fb_derevo_vidpochynok1_send(str_Rec:=fb_KL6301_0.str_Data_Rec, bData:=derevo_vidpochynok1,  Group_Address:=derevo_vidpochynok1_adr, bsend:=((fb_derevo_vidpochynok1_send.bData XOR fb_derevo_vidpochynok1_read.bData XOR derevo_vidpochynok1)OR fb_heartbeat_derevo_timer.q));
IF NOT fb_derevo_vidpochynok1_read.bDataReceive OR  EIB.fb_heartbeat_derevo_timer.q THEN fb_derevo_vidpochynok1_send.bSend:=FALSE; fb_derevo_vidpochynok1_send(str_Rec:=fb_KL6301_0.str_Data_Rec, bData:=derevo_vidpochynok1,  Group_Address:=derevo_vidpochynok1_adr);END_IF
fb_derevo_vidpochynok2_send(str_Rec:=fb_KL6301_0.str_Data_Rec, bData:=derevo_vidpochynok2,  Group_Address:=derevo_vidpochynok2_adr, bsend:=((fb_derevo_vidpochynok2_send.bData XOR fb_derevo_vidpochynok2_read.bData XOR derevo_vidpochynok2)OR fb_heartbeat_derevo_timer.q));
IF NOT fb_derevo_vidpochynok2_read.bDataReceive OR  fb_heartbeat_derevo_timer.q THEN fb_derevo_vidpochynok2_send.bSend:=FALSE; fb_derevo_vidpochynok2_send(str_Rec:=fb_KL6301_0.str_Data_Rec, bData:=derevo_vidpochynok2,  Group_Address:=derevo_vidpochynok2_adr);END_IF
fb_derevo_veranda_send(str_Rec:=fb_KL6301_0.str_Data_Rec, bData:=derevo_veranda,  Group_Address:=derevo_veranda_adr, bsend:=((fb_derevo_veranda_send.bData XOR fb_derevo_veranda_read.bData XOR derevo_veranda)OR fb_heartbeat_derevo_timer.q));
IF NOT fb_derevo_veranda_read.bDataReceive OR  fb_heartbeat_derevo_timer.q THEN fb_derevo_veranda_send.bSend:=FALSE; fb_derevo_veranda_send(str_Rec:=fb_KL6301_0.str_Data_Rec, bData:=derevo_veranda,  Group_Address:=derevo_veranda_adr);END_IF
fb_derevo_veranda_zovn_send(str_Rec:=fb_KL6301_0.str_Data_Rec, bData:=derevo_veranda_zovn,  Group_Address:=derevo_veranda_zovn_adr, bsend:=((fb_derevo_veranda_zovn_send.bData XOR fb_derevo_veranda_zovn_read.bData XOR derevo_veranda_zovn)OR fb_heartbeat_derevo_timer.q));
IF NOT fb_derevo_veranda_zovn_read.bDataReceive OR  fb_heartbeat_derevo_timer.q THEN fb_derevo_veranda_zovn_send.bSend:=FALSE; fb_derevo_veranda_zovn_send(str_Rec:=fb_KL6301_0.str_Data_Rec, bData:=derevo_veranda_zovn,  Group_Address:=derevo_veranda_zovn_adr);END_IF
fb_derevo_vhid_zovn_send(str_Rec:=fb_KL6301_0.str_Data_Rec, bData:=derevo_vhid_zovn,  Group_Address:=derevo_vhid_zovn_adr, bsend:=((fb_derevo_vhid_zovn_send.bData XOR fb_derevo_vhid_zovn_read.bData XOR derevo_vhid_zovn)OR fb_heartbeat_derevo_timer.q));
IF NOT fb_derevo_vhid_zovn_read.bDataReceive OR  fb_heartbeat_derevo_timer.q THEN fb_derevo_vhid_zovn_send.bSend:=FALSE; fb_derevo_vhid_zovn_send(str_Rec:=fb_KL6301_0.str_Data_Rec, bData:=derevo_vhid_zovn,  Group_Address:=derevo_vhid_zovn_adr);END_IF
fb_derevo_sauna_send(str_Rec:=fb_KL6301_0.str_Data_Rec, bData:=derevo_sauna,  Group_Address:=derevo_sauna_adr, bsend:=((fb_derevo_sauna_send.bData XOR fb_derevo_sauna_read.bData XOR derevo_sauna)OR fb_heartbeat_derevo_timer.q));
IF NOT fb_derevo_sauna_read.bDataReceive OR  fb_heartbeat_derevo_timer.q THEN fb_derevo_sauna_send.bSend:=FALSE; fb_derevo_sauna_send(str_Rec:=fb_KL6301_0.str_Data_Rec, bData:=derevo_sauna,  Group_Address:=derevo_sauna_adr);END_IF
fb_derevo_vhid_send(str_Rec:=fb_KL6301_0.str_Data_Rec, bData:=derevo_vhid,  Group_Address:=derevo_vhid_adr, bsend:=((fb_derevo_vhid_send.bData XOR fb_derevo_vhid_read.bData XOR derevo_vhid)OR fb_heartbeat_derevo_timer.q));
IF NOT fb_derevo_vhid_read.bDataReceive OR  fb_heartbeat_derevo_timer.q THEN fb_derevo_vhid_send.bSend:=FALSE; fb_derevo_vhid_send(str_Rec:=fb_KL6301_0.str_Data_Rec, bData:=derevo_vhid,  Group_Address:=derevo_vhid_adr);END_IF
fb_derevo_kotel_send(str_Rec:=fb_KL6301_0.str_Data_Rec, bData:=derevo_kotel,  Group_Address:=derevo_kotel_adr, bsend:=((fb_derevo_kotel_send.bData XOR fb_derevo_kotel_read.bData XOR derevo_kotel)OR fb_heartbeat_derevo_timer.q));
IF NOT fb_derevo_kotel_read.bDataReceive OR  fb_heartbeat_derevo_timer.q THEN fb_derevo_kotel_send.bSend:=FALSE; fb_derevo_kotel_send(str_Rec:=fb_KL6301_0.str_Data_Rec, bData:=derevo_kotel,  Group_Address:=derevo_kotel_adr);END_IF
fb_derevo_korydor_send(str_Rec:=fb_KL6301_0.str_Data_Rec, bData:=derevo_korydor,  Group_Address:=derevo_korydor_adr, bsend:=((fb_derevo_korydor_send.bData XOR fb_derevo_korydor_read.bData XOR derevo_korydor)OR fb_heartbeat_derevo_timer.q));
IF NOT fb_derevo_korydor_read.bDataReceive OR  fb_heartbeat_derevo_timer.q THEN fb_derevo_korydor_send.bSend:=FALSE; fb_derevo_korydor_send(str_Rec:=fb_KL6301_0.str_Data_Rec, bData:=derevo_korydor,  Group_Address:=derevo_korydor_adr);END_IF
fb_derevo_sinna_send(str_Rec:=fb_KL6301_0.str_Data_Rec, bData:=derevo_sinna,  Group_Address:=derevo_sinna_adr, bsend:=((fb_derevo_sinna_send.bData XOR fb_derevo_sinna_read.bData XOR derevo_sinna)OR fb_heartbeat_derevo_timer.q));
IF NOT fb_derevo_sinna_read.bDataReceive OR  fb_heartbeat_derevo_timer.q THEN fb_derevo_sinna_send.bSend:=FALSE; fb_derevo_sinna_send(str_Rec:=fb_KL6301_0.str_Data_Rec, bData:=derevo_sinna,  Group_Address:=derevo_sinna_adr);END_IF
fb_derevo_hamam_send(str_Rec:=fb_KL6301_0.str_Data_Rec, bData:=derevo_hamam,  Group_Address:=derevo_hamam_adr, bsend:=((fb_derevo_hamam_send.bData XOR fb_derevo_hamam_read.bData XOR derevo_hamam)OR fb_heartbeat_derevo_timer.q));
IF NOT fb_derevo_hamam_read.bDataReceive OR  fb_heartbeat_derevo_timer.q THEN fb_derevo_hamam_send.bSend:=FALSE; fb_derevo_hamam_send(str_Rec:=fb_KL6301_0.str_Data_Rec, bData:=derevo_hamam,  Group_Address:=derevo_hamam_adr);END_IF
fb_derevo_kuhnya_send(str_Rec:=fb_KL6301_0.str_Data_Rec, bData:=derevo_kuhnya,  Group_Address:=derevo_kuhnya_adr, bsend:=((fb_derevo_kuhnya_send.bData XOR fb_derevo_kuhnya_read.bData XOR derevo_kuhnya)OR fb_heartbeat_derevo_timer.q));
IF NOT fb_derevo_kuhnya_read.bDataReceive OR  fb_heartbeat_derevo_timer.q THEN fb_derevo_kuhnya_send.bSend:=FALSE; fb_derevo_kuhnya_send(str_Rec:=fb_KL6301_0.str_Data_Rec, bData:=derevo_kuhnya,  Group_Address:=derevo_kuhnya_adr);END_IF
fb_derevo_bassein1_send(str_Rec:=fb_KL6301_0.str_Data_Rec, bData:=derevo_bassein1,  Group_Address:=derevo_bassein1_adr, bsend:=((fb_derevo_bassein1_send.bData XOR fb_derevo_bassein1_read.bData XOR derevo_bassein1)OR fb_heartbeat_derevo_timer.q));
IF NOT fb_derevo_bassein1_read.bDataReceive OR  fb_heartbeat_derevo_timer.q THEN fb_derevo_bassein1_send.bSend:=FALSE; fb_derevo_bassein1_send(str_Rec:=fb_KL6301_0.str_Data_Rec, bData:=derevo_bassein1,  Group_Address:=derevo_bassein1_adr);END_IF
fb_derevo_bassein2_send(str_Rec:=fb_KL6301_0.str_Data_Rec, bData:=derevo_bassein2,  Group_Address:=derevo_bassein2_adr, bsend:=((fb_derevo_bassein2_send.bData XOR fb_derevo_bassein2_read.bData XOR derevo_bassein2)OR fb_heartbeat_derevo_timer.q));
IF NOT fb_derevo_bassein2_read.bDataReceive OR  fb_heartbeat_derevo_timer.q THEN fb_derevo_bassein2_send.bSend:=FALSE; fb_derevo_bassein2_send(str_Rec:=fb_KL6301_0.str_Data_Rec, bData:=derevo_bassein2,  Group_Address:=derevo_bassein2_adr);END_IF
fb_derevo_spalnya2_send(str_Rec:=fb_KL6301_0.str_Data_Rec, bData:=derevo_spalnya2,  Group_Address:=derevo_spalnya2_adr, bsend:=((fb_derevo_spalnya2_send.bData XOR fb_derevo_spalnya2_read.bData XOR derevo_spalnya2)OR fb_heartbeat_derevo_timer.q));
IF NOT fb_derevo_spalnya2_read.bDataReceive OR  fb_heartbeat_derevo_timer.q THEN fb_derevo_spalnya2_send.bSend:=FALSE; fb_derevo_spalnya2_send(str_Rec:=fb_KL6301_0.str_Data_Rec, bData:=derevo_spalnya2,  Group_Address:=derevo_spalnya2_adr);END_IF
fb_derevo_terassa_send(str_Rec:=fb_KL6301_0.str_Data_Rec, bData:=derevo_terassa,  Group_Address:=derevo_terassa_adr, bsend:=((fb_derevo_terassa_send.bData XOR fb_derevo_terassa_read.bData XOR derevo_terassa)OR fb_heartbeat_derevo_timer.q));
IF NOT fb_derevo_terassa_read.bDataReceive OR  fb_heartbeat_derevo_timer.q THEN fb_derevo_terassa_send.bSend:=FALSE; fb_derevo_terassa_send(str_Rec:=fb_KL6301_0.str_Data_Rec, bData:=derevo_terassa,  Group_Address:=derevo_terassa_adr);END_IF
fb_derevo_dush_send(str_Rec:=fb_KL6301_0.str_Data_Rec, bData:=derevo_dush,  Group_Address:=derevo_dush_adr, bsend:=((fb_derevo_dush_send.bData XOR fb_derevo_dush_read.bData XOR derevo_dush)OR fb_heartbeat_derevo_timer.q));
IF NOT fb_derevo_dush_read.bDataReceive OR  fb_heartbeat_derevo_timer.q THEN fb_derevo_dush_send.bSend:=FALSE; fb_derevo_dush_send(str_Rec:=fb_KL6301_0.str_Data_Rec, bData:=derevo_dush,  Group_Address:=derevo_dush_adr);END_IF
fb_derevo_wc_send(str_Rec:=fb_KL6301_0.str_Data_Rec, bData:=derevo_wc,  Group_Address:=derevo_wc_adr, bsend:=((fb_derevo_wc_send.bData XOR fb_derevo_wc_read.bData XOR derevo_wc)OR fb_heartbeat_derevo_timer.q));
IF NOT fb_derevo_wc_read.bDataReceive OR  fb_heartbeat_derevo_timer.q THEN fb_derevo_wc_send.bSend:=FALSE; fb_derevo_wc_send(str_Rec:=fb_KL6301_0.str_Data_Rec, bData:=derevo_wc,  Group_Address:=derevo_wc_adr);END_IF
fb_derevo_spalnya_verh_send(str_Rec:=fb_KL6301_0.str_Data_Rec, bData:=derevo_spalnya_verh,  Group_Address:=derevo_spalnya_verh_adr, bsend:=((fb_derevo_spalnya_verh_send.bData XOR fb_derevo_spalnya_verh_read.bData XOR derevo_spalnya_verh)OR fb_heartbeat_derevo_timer.q));
IF NOT fb_derevo_spalnya_verh_read.bDataReceive OR  fb_heartbeat_derevo_timer.q THEN fb_derevo_spalnya_verh_send.bSend:=FALSE; fb_derevo_spalnya_verh_send(str_Rec:=fb_KL6301_0.str_Data_Rec, bData:=derevo_spalnya_verh,  Group_Address:=derevo_spalnya_verh_adr);END_IF
fb_derevo_spalnya1_send(str_Rec:=fb_KL6301_0.str_Data_Rec, bData:=derevo_spalnya1,  Group_Address:=derevo_spalnya1_adr, bsend:=((fb_derevo_spalnya1_send.bData XOR fb_derevo_spalnya1_read.bData XOR derevo_spalnya1)OR fb_heartbeat_derevo_timer.q));
IF NOT fb_derevo_spalnya1_read.bDataReceive OR  fb_heartbeat_derevo_timer.q THEN fb_derevo_spalnya1_send.bSend:=FALSE; fb_derevo_spalnya1_send(str_Rec:=fb_KL6301_0.str_Data_Rec, bData:=derevo_spalnya1,  Group_Address:=derevo_spalnya1_adr);END_IF
fb_derevo_spalnya_su_send(str_Rec:=fb_KL6301_0.str_Data_Rec, bData:=derevo_spalnya_su,  Group_Address:=derevo_spalnya_su_adr, bsend:=((fb_derevo_spalnya_su_send.bData XOR fb_derevo_spalnya_su_read.bData XOR derevo_spalnya_su)OR fb_heartbeat_derevo_timer.q));
IF NOT fb_derevo_spalnya_su_read.bDataReceive OR  fb_heartbeat_derevo_timer.q THEN fb_derevo_spalnya_su_send.bSend:=FALSE; fb_derevo_spalnya_su_send(str_Rec:=fb_KL6301_0.str_Data_Rec, bData:=derevo_spalnya_su,  Group_Address:=derevo_spalnya_su_adr);END_IF
fb_derevo_garderob_send(str_Rec:=fb_KL6301_0.str_Data_Rec, bData:=derevo_garderob,  Group_Address:=derevo_garderob_adr, bsend:=((fb_derevo_garderob_send.bData XOR fb_derevo_garderob_read.bData XOR derevo_garderob)OR fb_heartbeat_derevo_timer.q));
IF NOT fb_derevo_garderob_read.bDataReceive OR  fb_heartbeat_derevo_timer.q THEN fb_derevo_garderob_send.bSend:=FALSE; fb_derevo_garderob_send(str_Rec:=fb_KL6301_0.str_Data_Rec, bData:=derevo_garderob,  Group_Address:=derevo_garderob_adr);END_IF

IF NOT fb_derevo_vidpochynok1_read.bDataReceive THEN
	data_derevo[100].0:= fb_derevo_vidpochynok1_read.bdata;
	derevo_vidpochynok1:= fb_derevo_vidpochynok1_read.bdata;
ELSE data_derevo[100].0:= derevo_vidpochynok1;END_IF
IF NOT fb_derevo_vidpochynok2_read.bDataReceive THEN
	data_derevo[100].1:= fb_derevo_vidpochynok2_read.bdata;
	derevo_vidpochynok2:= fb_derevo_vidpochynok2_read.bdata;
ELSE data_derevo[100].1:= derevo_vidpochynok2;END_IF
IF NOT fb_derevo_veranda_read.bDataReceive THEN
	data_derevo[100].2:= fb_derevo_veranda_read.bdata;
	derevo_veranda:= fb_derevo_veranda_read.bdata;
ELSE data_derevo[100].2:= derevo_veranda;END_IF
IF NOT fb_derevo_veranda_zovn_read.bDataReceive THEN
	data_derevo[100].3:= fb_derevo_veranda_zovn_read.bdata;
	derevo_veranda_zovn:= fb_derevo_veranda_zovn_read.bdata;
ELSE data_derevo[100].3:= derevo_veranda_zovn;END_IF
IF NOT fb_derevo_vhid_zovn_read.bDataReceive THEN
	data_derevo[100].4:= fb_derevo_vhid_zovn_read.bdata;
	derevo_vhid_zovn:= fb_derevo_vhid_zovn_read.bdata;
ELSE data_derevo[100].4:= derevo_vhid_zovn;END_IF
IF NOT fb_derevo_sauna_read.bDataReceive THEN
	data_derevo[100].5:= fb_derevo_sauna_read.bdata;
	derevo_sauna:= fb_derevo_sauna_read.bdata;
ELSE data_derevo[100].5:= derevo_sauna;END_IF
IF NOT fb_derevo_vhid_read.bDataReceive THEN
	data_derevo[100].6:= fb_derevo_vhid_read.bdata;
	derevo_vhid:= fb_derevo_vhid_read.bdata;
ELSE data_derevo[100].6:= derevo_vhid;END_IF
IF NOT fb_derevo_kotel_read.bDataReceive THEN
	data_derevo[100].7:= fb_derevo_kotel_read.bdata;
	derevo_kotel:= fb_derevo_kotel_read.bdata;
ELSE data_derevo[100].7:= derevo_kotel;END_IF
IF NOT fb_derevo_korydor_read.bDataReceive THEN
	data_derevo[101].0:= fb_derevo_korydor_read.bdata;
	derevo_korydor:= fb_derevo_korydor_read.bdata;
ELSE data_derevo[101].0:= derevo_korydor;END_IF
IF NOT fb_derevo_sinna_read.bDataReceive THEN
	data_derevo[101].1:= fb_derevo_sinna_read.bdata;
	derevo_sinna:= fb_derevo_sinna_read.bdata;
ELSE data_derevo[101].1:= derevo_sinna;END_IF
IF NOT fb_derevo_hamam_read.bDataReceive THEN
	data_derevo[101].2:= fb_derevo_hamam_read.bdata;
	derevo_hamam:= fb_derevo_hamam_read.bdata;
ELSE data_derevo[101].2:= derevo_hamam;END_IF
IF NOT fb_derevo_kuhnya_read.bDataReceive THEN
	data_derevo[101].3:= fb_derevo_kuhnya_read.bdata;
	derevo_kuhnya:= fb_derevo_kuhnya_read.bdata;
ELSE data_derevo[101].3:= derevo_kuhnya;END_IF
IF NOT fb_derevo_bassein1_read.bDataReceive THEN
	data_derevo[101].4:= fb_derevo_bassein1_read.bdata;
	derevo_bassein1:= fb_derevo_bassein1_read.bdata;
ELSE data_derevo[101].4:= derevo_bassein1;END_IF
IF NOT fb_derevo_bassein2_read.bDataReceive THEN
	data_derevo[101].5:= fb_derevo_bassein2_read.bdata;
	derevo_bassein2:= fb_derevo_bassein2_read.bdata;
ELSE data_derevo[101].5:= derevo_bassein2;END_IF
IF NOT fb_derevo_spalnya2_read.bDataReceive THEN
	data_derevo[101].6:= fb_derevo_spalnya2_read.bdata;
	derevo_spalnya2:= fb_derevo_spalnya2_read.bdata;
ELSE data_derevo[101].6:= derevo_spalnya2;END_IF
IF NOT fb_derevo_terassa_read.bDataReceive THEN
	data_derevo[101].7:= fb_derevo_terassa_read.bdata;
	derevo_terassa:= fb_derevo_terassa_read.bdata;
ELSE data_derevo[101].7:= derevo_terassa;END_IF
IF NOT fb_derevo_dush_read.bDataReceive THEN
	data_derevo[102].0:= fb_derevo_dush_read.bdata;
	derevo_dush:= fb_derevo_dush_read.bdata;
ELSE data_derevo[102].0:= derevo_dush;END_IF
IF NOT fb_derevo_wc_read.bDataReceive THEN
	data_derevo[102].1:= fb_derevo_wc_read.bdata;
	derevo_wc:= fb_derevo_wc_read.bdata;
ELSE data_derevo[102].1:= derevo_spalnya_verh;END_IF
IF NOT fb_derevo_spalnya_verh_read.bDataReceive THEN
	data_derevo[102].2:= fb_derevo_spalnya_verh_read.bdata;
	derevo_spalnya_verh:= fb_derevo_spalnya_verh_read.bdata;
ELSE data_derevo[102].2:= derevo_spalnya_verh;END_IF
IF NOT fb_derevo_spalnya1_read.bDataReceive THEN
	data_derevo[102].3:= fb_derevo_spalnya1_read.bdata;
	derevo_spalnya1:= fb_derevo_spalnya1_read.bdata;
ELSE data_derevo[102].3:= derevo_spalnya1;END_IF
IF NOT fb_derevo_spalnya_su_read.bDataReceive THEN
	data_derevo[102].4:= fb_derevo_spalnya_su_read.bdata;
	derevo_spalnya_su:= fb_derevo_spalnya_su_read.bdata;
ELSE data_derevo[102].4:= derevo_spalnya_su;END_IF
IF NOT fb_derevo_garderob_read.bDataReceive THEN
	data_derevo[102].5:= fb_derevo_garderob_read.bdata;
	derevo_garderob:= fb_derevo_garderob_read.bdata;
ELSE data_derevo[102].5:= derevo_garderob;END_IF
END_ACTION
ACTION floor1:
fb_komora_l_read(strData_Rec:=fb_KL6301_0.str_Data_Rec,   Group_Address:=komora_l_adr);
fb_su1_l_read(strData_Rec:=fb_KL6301_0.str_Data_Rec,   Group_Address:=su1_l_adr);
fb_topochna_l_read(strData_Rec:=fb_KL6301_0.str_Data_Rec,  Group_Address:=topochna_l_adr);
fb_su2_bra_read(strData_Rec:=fb_KL6301_0.str_Data_Rec, Group_Address:=su2_bra_adr);
fb_topochna2_l_read(strData_Rec:=fb_KL6301_0.str_Data_Rec, Group_Address:=topochna2_l_adr);
fb_su2_l_read(strData_Rec:=fb_KL6301_0.str_Data_Rec, Group_Address:=su2_l_adr);
fb_su1_rakovyna_read(strData_Rec:=fb_KL6301_0.str_Data_Rec, Group_Address:=su1_rakovyna_adr);
fb_dush_read(strData_Rec:=fb_KL6301_0.str_Data_Rec, Group_Address:=dush_adr);
fb_su2_dush_read(strData_Rec:=fb_KL6301_0.str_Data_Rec, Group_Address:=su2_dush_adr);
fb_vitalnya_smugy2_read(strData_Rec:=fb_KL6301_0.str_Data_Rec, Group_Address:=vitalnya_smugy2_adr);
fb_su2_polytsi_read(strData_Rec:=fb_KL6301_0.str_Data_Rec, Group_Address:=su2_polytsi_adr);
fb_kuhnya1_read(strData_Rec:=fb_KL6301_0.str_Data_Rec, Group_Address:=kuhnya1_adr);
fb_kuhnya2_read(strData_Rec:=fb_KL6301_0.str_Data_Rec, Group_Address:=kuhnya2_adr);
fb_vitalnya_smugy1_read(strData_Rec:=fb_KL6301_0.str_Data_Rec, Group_Address:=vitalnya_smugy1_adr);
fb_vitalnya_l_read(strData_Rec:=fb_KL6301_0.str_Data_Rec, Group_Address:=vitalnya_l_adr);
fb_vitalnya_prokladka_read(strData_Rec:=fb_KL6301_0.str_Data_Rec, Group_Address:=vitalnya_prokladka_adr);
fb_terassa_stina_read(strData_Rec:=fb_KL6301_0.str_Data_Rec, Group_Address:=terassa_stina_adr);
fb_pidval_shody_read(strData_Rec:=fb_KL6301_0.str_Data_Rec, Group_Address:=pidval_shody_adr);
fb_terassa_read(strData_Rec:=fb_KL6301_0.str_Data_Rec, Group_Address:=terassa_adr);
fb_skhody2pov_read(strData_Rec:=fb_KL6301_0.str_Data_Rec, Group_Address:=skhody2pov_adr);
fb_tambur_l_read(strData_Rec:=fb_KL6301_0.str_Data_Rec, Group_Address:=tambur_l_adr);

fb_komora_l_send(str_Rec:=fb_KL6301_0.str_Data_Rec, bData:=komora_l,  Group_Address:=komora_l_adr, bsend:=((fb_komora_l_send.bData XOR fb_komora_l_read.bData XOR komora_l  )OR fb_heartbeat_timer.q))      ;
IF NOT fb_komora_l_read.bDataReceive OR  fb_heartbeat1_timer.q THEN fb_komora_l_send.bSend:=FALSE; fb_komora_l_send(str_Rec:=fb_KL6301_0.str_Data_Rec, bData:=komora_l,  Group_Address:=komora_l_adr);END_IF
fb_su1_l_send(str_Rec:=fb_KL6301_0.str_Data_Rec, bData:=su1_l,  Group_Address:=su1_l_adr, bsend:=(fb_su1_l_read.bData XOR (fb_su1_l_read.bData XOR su1_l)OR fb_heartbeat1_timer.q))      ;
IF NOT fb_su1_l_read.bDataReceive OR  fb_heartbeat1_timer.q THEN fb_su1_l_send.bSend:=FALSE; fb_su1_l_send(str_Rec:=fb_KL6301_0.str_Data_Rec, bData:=su1_l,  Group_Address:=su1_l_adr);END_IF
fb_topochna_l_send(str_Rec:=fb_KL6301_0.str_Data_Rec, bData:=topochna_l,  Group_Address:=topochna_l_adr, bsend:=((fb_topochna_l_send.bData XOR fb_topochna_l_read.bData XOR topochna_l)OR fb_heartbeat1_timer.q))      ;
IF NOT fb_topochna_l_read.bDataReceive OR  fb_heartbeat1_timer.q THEN fb_topochna_l_send.bSend:=FALSE; fb_topochna_l_send(str_Rec:=fb_KL6301_0.str_Data_Rec, bData:=topochna_l,  Group_Address:=topochna_l_adr);END_IF
fb_su2_bra_send(str_Rec:=fb_KL6301_0.str_Data_Rec, bData:=su2_bra,  Group_Address:=su2_bra_adr, bsend:=((fb_su2_bra_read.bData  XOR fb_su2_bra_read.bData XOR su2_bra)OR fb_heartbeat1_timer.q))      ;
IF NOT fb_su2_bra_read.bDataReceive OR  fb_heartbeat1_timer.q THEN fb_su2_bra_send.bSend:=FALSE; fb_su2_bra_send(str_Rec:=fb_KL6301_0.str_Data_Rec, bData:=su2_bra,  Group_Address:=su2_bra_adr);END_IF
fb_topochna2_l_send(str_Rec:=fb_KL6301_0.str_Data_Rec, bData:=topochna2_l,  Group_Address:=topochna2_l_adr, bsend:=((fb_topochna2_l_send.bData XOR fb_topochna2_l_read.bData XOR topochna2_l)OR fb_heartbeat1_timer.q))      ;
IF NOT fb_topochna2_l_read.bDataReceive OR  fb_heartbeat1_timer.q THEN fb_topochna2_l_send.bSend:=FALSE; fb_topochna2_l_send(str_Rec:=fb_KL6301_0.str_Data_Rec, bData:=topochna2_l,  Group_Address:=topochna2_l_adr);END_IF
fb_su2_l_send(str_Rec:=fb_KL6301_0.str_Data_Rec, bData:=su2_l,  Group_Address:=su2_l_adr, bsend:=((fb_su2_l_read.bData  XOR fb_su2_l_read.bData XOR su2_l)OR fb_heartbeat1_timer.q))      ;
IF NOT fb_su2_l_read.bDataReceive OR  fb_heartbeat1_timer.q THEN fb_su2_l_send.bSend:=FALSE; fb_su2_l_send(str_Rec:=fb_KL6301_0.str_Data_Rec, bData:=su2_l,  Group_Address:=su2_l_adr);END_IF
fb_su1_rakovyna_send(str_Rec:=fb_KL6301_0.str_Data_Rec, bData:=su1_rakovyna,  Group_Address:=su1_rakovyna_adr, bsend:=((fb_su1_rakovyna_send.bData XOR fb_su1_rakovyna_read.bData XOR su1_rakovyna)OR fb_heartbeat1_timer.q))      ;
IF NOT fb_su1_rakovyna_read.bDataReceive OR  fb_heartbeat1_timer.q THEN fb_su1_rakovyna_send.bSend:=FALSE; fb_su1_rakovyna_send(str_Rec:=fb_KL6301_0.str_Data_Rec, bData:=su1_rakovyna,  Group_Address:=su1_rakovyna_adr);END_IF
fb_su2_dush_send(str_Rec:=fb_KL6301_0.str_Data_Rec, bData:=su2_dush,  Group_Address:=su2_dush_adr, bsend:=((fb_su2_dush_send.bData XOR fb_su2_dush_read.bData XOR su2_dush)OR fb_heartbeat1_timer.q))      ;
IF NOT fb_su2_dush_read.bDataReceive OR  fb_heartbeat1_timer.q THEN fb_su2_dush_send.bSend:=FALSE; fb_su2_dush_send(str_Rec:=fb_KL6301_0.str_Data_Rec, bData:=su2_dush,  Group_Address:=su2_dush_adr);END_IF
fb_dush_send(str_Rec:=fb_KL6301_0.str_Data_Rec, bData:=dush,  Group_Address:=dush_adr, bsend:=((fb_dush_send.bData XOR fb_dush_read.bData XOR dush)OR fb_heartbeat1_timer.q))      ;
IF NOT fb_dush_read.bDataReceive OR  fb_heartbeat1_timer.q THEN fb_dush_send.bSend:=FALSE; fb_dush_send(str_Rec:=fb_KL6301_0.str_Data_Rec, bData:=dush,  Group_Address:=dush_adr);END_IF
fb_vitalnya_smugy2_send(str_Rec:=fb_KL6301_0.str_Data_Rec, bData:=vitalnya_smugy2,  Group_Address:=vitalnya_smugy2_adr, bsend:=((fb_vitalnya_smugy2_send.bData XOR fb_vitalnya_smugy2_read.bData XOR vitalnya_smugy2)OR fb_heartbeat1_timer.q));   (*       vitalnya_smugy2_read.bData XOR vitalnya_smugy2)) AND fb_heartbeat1_timer.q))      )));*)
IF NOT fb_vitalnya_smugy2_read.bDataReceive OR  fb_heartbeat1_timer.q THEN fb_vitalnya_smugy2_send.bSend:=FALSE; fb_vitalnya_smugy2_send(str_Rec:=fb_KL6301_0.str_Data_Rec, bData:=vitalnya_smugy2,  Group_Address:=vitalnya_smugy2_adr);END_IF
fb_su2_polytsi_send(str_Rec:=fb_KL6301_0.str_Data_Rec, bData:=su2_polytsi,  Group_Address:=su2_polytsi_adr, bsend:=((fb_su2_polytsi_send.bData XOR fb_su2_polytsi_read.bData XOR su2_polytsi)OR fb_heartbeat1_timer.q));   (*       su2_polytsi_read.bData XOR su2_polytsi)) AND fb_heartbeat1_timer.q))      )));*)
IF NOT fb_su2_polytsi_read.bDataReceive OR  fb_heartbeat1_timer.q THEN fb_su2_polytsi_send.bSend:=FALSE; fb_su2_polytsi_send(str_Rec:=fb_KL6301_0.str_Data_Rec, bData:=su2_polytsi,  Group_Address:=su2_polytsi_adr);END_IF
fb_kuhnya1_send(str_Rec:=fb_KL6301_0.str_Data_Rec, bData:=kuhnya1,  Group_Address:=kuhnya1_adr, bsend:=((fb_kuhnya1_send.bData XOR fb_kuhnya1_read.bData XOR kuhnya1)OR fb_heartbeat1_timer.q));   (*       kuhnya1_read.bData XOR kuhnya1)) AND fb_heartbeat1_timer.q))      )));*)
IF NOT fb_kuhnya1_read.bDataReceive OR  fb_heartbeat1_timer.q THEN fb_kuhnya1_send.bSend:=FALSE; fb_kuhnya1_send(str_Rec:=fb_KL6301_0.str_Data_Rec, bData:=kuhnya1,  Group_Address:=kuhnya1_adr);END_IF
fb_kuhnya2_send(str_Rec:=fb_KL6301_0.str_Data_Rec, bData:=kuhnya2,  Group_Address:=kuhnya2_adr, bsend:=((fb_kuhnya2_send.bData XOR fb_kuhnya2_read.bData XOR kuhnya2)OR fb_heartbeat1_timer.q));   (*       kuhnya2_read.bData XOR kuhnya2)) AND fb_heartbeat1_timer.q))      )));*)
IF NOT fb_kuhnya2_read.bDataReceive OR  fb_heartbeat1_timer.q THEN fb_kuhnya2_send.bSend:=FALSE; fb_kuhnya2_send(str_Rec:=fb_KL6301_0.str_Data_Rec, bData:=kuhnya2,  Group_Address:=kuhnya2_adr);END_IF
fb_vitalnya_smugy1_send(str_Rec:=fb_KL6301_0.str_Data_Rec, bData:=vitalnya_smugy1,  Group_Address:=vitalnya_smugy1_adr, bsend:=((fb_vitalnya_smugy1_send.bData XOR fb_vitalnya_smugy1_read.bData XOR vitalnya_smugy1)OR fb_heartbeat1_timer.q));   (*       vitalnya_smugy1_read.bData XOR vitalnya_smugy1)) AND fb_heartbeat1_timer.q))      )));*)
IF NOT fb_vitalnya_smugy1_read.bDataReceive OR  fb_heartbeat1_timer.q THEN fb_vitalnya_smugy1_send.bSend:=FALSE; fb_vitalnya_smugy1_send(str_Rec:=fb_KL6301_0.str_Data_Rec, bData:=vitalnya_smugy1,  Group_Address:=vitalnya_smugy1_adr);END_IF
fb_vitalnya_l_send(str_Rec:=fb_KL6301_0.str_Data_Rec, bData:=vitalnya_l,  Group_Address:=vitalnya_l_adr, bsend:=((fb_vitalnya_l_send.bData XOR fb_vitalnya_l_read.bData XOR vitalnya_l)OR fb_heartbeat1_timer.q));   (*       vitalnya_l_read.bData XOR vitalnya_l)) AND fb_heartbeat1_timer.q))      )));*)
IF NOT fb_vitalnya_l_read.bDataReceive OR  fb_heartbeat1_timer.q THEN fb_vitalnya_l_send.bSend:=FALSE; fb_vitalnya_l_send(str_Rec:=fb_KL6301_0.str_Data_Rec, bData:=vitalnya_l,  Group_Address:=vitalnya_l_adr);END_IF
fb_vitalnya_prokladka_send(str_Rec:=fb_KL6301_0.str_Data_Rec, bData:=vitalnya_prokladka,  Group_Address:=vitalnya_prokladka_adr, bsend:=((fb_vitalnya_prokladka_send.bData XOR fb_vitalnya_prokladka_read.bData XOR vitalnya_prokladka)OR fb_heartbeat1_timer.q));   (*       vitalnya_prokladka_read.bData XOR vitalnya_prokladka)) AND fb_heartbeat1_timer.q))      )));*)
IF NOT fb_vitalnya_prokladka_read.bDataReceive OR  fb_heartbeat1_timer.q THEN fb_vitalnya_prokladka_send.bSend:=FALSE; fb_vitalnya_prokladka_send(str_Rec:=fb_KL6301_0.str_Data_Rec, bData:=vitalnya_prokladka,  Group_Address:=vitalnya_prokladka_adr);END_IF
fb_terassa_stina_send(str_Rec:=fb_KL6301_0.str_Data_Rec, bData:=terassa_stina,  Group_Address:=terassa_stina_adr, bsend:=((fb_terassa_stina_send.bData XOR fb_terassa_stina_read.bData XOR terassa_stina)OR fb_heartbeat1_timer.q));   (*       terassa_stina_read.bData XOR terassa_stina)) AND fb_heartbeat1_timer.q))      )));*)
IF NOT fb_terassa_stina_read.bDataReceive OR  fb_heartbeat1_timer.q THEN fb_terassa_stina_send.bSend:=FALSE; fb_terassa_stina_send(str_Rec:=fb_KL6301_0.str_Data_Rec, bData:=terassa_stina,  Group_Address:=terassa_stina_adr);END_IF
fb_pidval_shody_send(str_Rec:=fb_KL6301_0.str_Data_Rec, bData:=pidval_shody,  Group_Address:=pidval_shody_adr, bsend:=(fb_pidval_shody_read.bData  XOR (fb_pidval_shody_read.bData XOR pidval_shody)OR fb_heartbeat1_timer.q));   (*       pidval_shody_read.bData XOR pidval_shody)) AND fb_heartbeat1_timer.q))      )));*)
IF NOT fb_pidval_shody_read.bDataReceive OR  fb_heartbeat1_timer.q THEN fb_pidval_shody_send.bSend:=FALSE; fb_pidval_shody_send(str_Rec:=fb_KL6301_0.str_Data_Rec, bData:=pidval_shody,  Group_Address:=pidval_shody_adr);END_IF
fb_terassa_send(str_Rec:=fb_KL6301_0.str_Data_Rec, bData:=terassa,  Group_Address:=terassa_adr, bsend:=((fb_terassa_read.bData  XOR fb_terassa_read.bData XOR terassa)OR fb_heartbeat1_timer.q));   (*       terassa_read.bData XOR terassa)) AND fb_heartbeat1_timer.q))      )));*)
IF NOT fb_terassa_read.bDataReceive OR  fb_heartbeat1_timer.q THEN fb_terassa_send.bSend:=FALSE; fb_terassa_send(str_Rec:=fb_KL6301_0.str_Data_Rec, bData:=terassa,  Group_Address:=terassa_adr);END_IF
fb_skhody2pov_send(str_Rec:=fb_KL6301_0.str_Data_Rec, bData:=skhody2pov,  Group_Address:=skhody2pov_adr, bsend:=((fb_skhody2pov_send.bData XOR fb_skhody2pov_read.bData XOR skhody2pov)OR fb_heartbeat1_timer.q));   (*       skhody2pov_read.bData XOR skhody2pov)) AND fb_heartbeat1_timer.q))      )));*)
IF NOT fb_skhody2pov_read.bDataReceive OR  fb_heartbeat1_timer.q THEN fb_skhody2pov_send.bSend:=FALSE; fb_skhody2pov_send(str_Rec:=fb_KL6301_0.str_Data_Rec, bData:=skhody2pov,  Group_Address:=skhody2pov_adr);END_IF
fb_tambur_l_send(str_Rec:=fb_KL6301_0.str_Data_Rec, bData:=tambur_l,  Group_Address:=tambur_l_adr, bsend:=((fb_tambur_l_send.bData XOR fb_tambur_l_read.bData XOR tambur_l)OR fb_heartbeat1_timer.q));   (*       tambur_l_read.bData XOR tambur_l)) AND fb_heartbeat1_timer.q))      )));*)
IF NOT fb_tambur_l_read.bDataReceive OR  fb_heartbeat1_timer.q THEN fb_tambur_l_send.bSend:=FALSE; fb_tambur_l_send(str_Rec:=fb_KL6301_0.str_Data_Rec, bData:=tambur_l,  Group_Address:=tambur_l_adr);END_IF

IF NOT fb_komora_l_read.bDataReceive THEN
	data1floor[100].0:=fb_komora_l_read.bdata;
	komora_l:=fb_komora_l_read.bdata;
ELSE  data1floor[100].0:=komora_l; END_IF;
IF NOT fb_su1_l_read.bDataReceive THEN
	data1floor[100].1:=fb_su1_l_read.bdata;
	su1_l:=fb_su1_l_read.bdata;
ELSE  data1floor[100].1:=su1_l; END_IF;
IF NOT fb_topochna_l_read.bDataReceive THEN
	data1floor[100].2:=fb_topochna_l_read.bdata;
	topochna_l:=fb_topochna_l_read.bdata;
ELSE  data1floor[100].2:=topochna_l; END_IF;
IF NOT fb_su2_bra_read.bDataReceive THEN
	data1floor[100].3:=fb_su2_bra_read.bdata;
	su2_bra:=fb_su2_bra_read.bdata;
ELSE  data1floor[100].3:=su2_bra; END_IF;
IF NOT fb_topochna2_l_read.bDataReceive THEN
	data1floor[100].4:=fb_topochna2_l_read.bdata;
	topochna2_l:=fb_topochna2_l_read.bdata;
ELSE  data1floor[100].4:=topochna2_l; END_IF;
IF NOT fb_su2_l_read.bDataReceive  THEN
	data1floor[100].5:=fb_su2_l_read.bdata;
	su2_l:=fb_su2_l_read.bdata;
ELSE  data1floor[100].5:=su2_l; END_IF;
IF NOT fb_su1_rakovyna_read.bDataReceive THEN
	data1floor[100].6:=fb_su1_rakovyna_read.bdata;
	su1_rakovyna:=fb_su1_rakovyna_read.bdata;
ELSE  data1floor[100].6:=su1_rakovyna; END_IF;
IF NOT fb_su2_dush_read.bDataReceive THEN
	data1floor[100].7:=fb_su2_dush_read.bdata;
	su2_dush:=fb_su2_dush_read.bdata;
ELSE  data1floor[100].7:=su2_dush; END_IF;
IF NOT fb_dush_read.bDataReceive  THEN
	data1floor[101].0:=fb_dush_read.bdata;
	dush:=fb_dush_read.bdata;
ELSE  data1floor[101].0:=dush; END_IF;
IF NOT fb_vitalnya_smugy2_read.bDataReceive THEN
	data1floor[101].1:=fb_vitalnya_smugy2_read.bdata;
	vitalnya_smugy2:=fb_vitalnya_smugy2_read.bdata;
ELSE  data1floor[101].1:=vitalnya_smugy2; END_IF;
IF NOT fb_su2_polytsi_read.bDataReceive  THEN
	data1floor[101].2:=fb_su2_polytsi_read.bdata;
	su2_polytsi:=fb_su2_polytsi_read.bdata;
ELSE  data1floor[101].2:=su2_polytsi; END_IF;
IF NOT fb_kuhnya1_read.bDataReceive  THEN
	data1floor[101].3:=fb_kuhnya1_read.bdata;
	kuhnya1:=fb_kuhnya1_read.bdata;
ELSE  data1floor[101].3:=kuhnya1; END_IF;
IF NOT fb_kuhnya2_read.bDataReceive  THEN
	data1floor[101].4:=fb_kuhnya2_read.bdata;
	kuhnya2:=fb_kuhnya2_read.bdata;
ELSE  data1floor[101].4:=kuhnya2; END_IF;
IF NOT fb_vitalnya_smugy1_read.bDataReceive THEN
	data1floor[101].5:=fb_vitalnya_smugy1_read.bdata;
	vitalnya_smugy1:=fb_vitalnya_smugy1_read.bdata;
ELSE  data1floor[101].5:=vitalnya_smugy1; END_IF;
IF NOT fb_vitalnya_l_read.bDataReceive  THEN
	data1floor[101].6:=fb_vitalnya_l_read.bdata;
	vitalnya_l:=fb_vitalnya_l_read.bdata;
ELSE  data1floor[101].6:=vitalnya_l; END_IF;
IF NOT fb_vitalnya_prokladka_read.bDataReceive  THEN
	data1floor[101].7:=fb_vitalnya_prokladka_read.bdata;
	vitalnya_prokladka:=fb_vitalnya_prokladka_read.bdata;
ELSE  data1floor[101].7:=vitalnya_prokladka; END_IF;
IF NOT fb_terassa_stina_read.bDataReceive THEN
	data1floor[102].0:=fb_terassa_stina_read.bdata;
	terassa_stina:=fb_terassa_stina_read.bdata;
 ELSE  data1floor[102].0:=terassa_stina; END_IF;
IF NOT fb_pidval_shody_read.bDataReceive  THEN
	data1floor[102].1:=fb_pidval_shody_read.bdata;
	pidval_shody:=fb_pidval_shody_read.bdata;
ELSE  data1floor[102].1:=pidval_shody; END_IF;
IF NOT fb_terassa_read.bDataReceive  THEN
	data1floor[102].2:=fb_terassa_read.bdata;
	terassa:=fb_terassa_read.bdata;
ELSE data1floor[102].2:=terassa; END_IF;
IF NOT fb_skhody2pov_read.bDataReceive THEN
	data1floor[102].3:=fb_skhody2pov_read.bdata;
	skhody2pov:=fb_skhody2pov_read.bdata;
 ELSE  data1floor[102].3:=skhody2pov; END_IF;
IF NOT fb_tambur_l_read.bDataReceive  THEN
	data1floor[102].4:=fb_tambur_l_read.bdata;
	tambur_l:=fb_tambur_l_read.bdata;
ELSE  data1floor[102].4:=tambur_l; END_IF;
END_ACTION
ACTION floor2:
fb_balkon_peryla_read(strData_Rec:=fb_KL6301_0.str_Data_Rec, Group_Address:=balkon_peryla_adr);
fb_kino_l_read(strData_Rec:=fb_KL6301_0.str_Data_Rec, Group_Address:=kino_l_adr);
fb_balkon_bra_read(strData_Rec:=fb_KL6301_0.str_Data_Rec, Group_Address:=balkon_bra_adr);
fb_kabinet_balkon_l_read(strData_Rec:=fb_KL6301_0.str_Data_Rec, Group_Address:=kabinet_balkon_l_adr);
fb_balkon_read(strData_Rec:=fb_KL6301_0.str_Data_Rec, Group_Address:=balkon_adr);
fb_korydor1_read(strData_Rec:=fb_KL6301_0.str_Data_Rec, Group_Address:=korydor1_adr);
fb_kino_bra_read(strData_Rec:=fb_KL6301_0.str_Data_Rec, Group_Address:=kino_bra_adr);
fb_korydor2_read(strData_Rec:=fb_KL6301_0.str_Data_Rec,  Group_Address:=korydor2_adr);
fb_studio_pidsvitka_read(strData_Rec:=fb_KL6301_0.str_Data_Rec, Group_Address:=studio_pidsvitka_adr);
fb_skhody2_3_read(strData_Rec:=fb_KL6301_0.str_Data_Rec, Group_Address:=skhody2_3_adr);
fb_studio_l_read(strData_Rec:=fb_KL6301_0.str_Data_Rec, Group_Address:=studio_l_adr);
fb_kabinet_pidsvitka_kolo_read(strData_Rec:=fb_KL6301_0.str_Data_Rec, Group_Address:=kabinet_pidsvitka_kolo_adr);
fb_kabinet_svitlo_read(strData_Rec:=fb_KL6301_0.str_Data_Rec, Group_Address:=kabinet_svitlo_adr);
fb_stend_read(strData_Rec:=fb_KL6301_0.str_Data_Rec, Group_Address:=stend_adr);
fb_kabinet_kobra_read(strData_Rec:=fb_KL6301_0.str_Data_Rec, Group_Address:=kabinet_kobra_adr);
fb_skhody_peryla_read(strData_Rec:=fb_KL6301_0.str_Data_Rec,Group_Address:=skhody_peryla_adr);
fb_tambur2_read(strData_Rec:=fb_KL6301_0.str_Data_Rec, Group_Address:=tambur2_adr);

fb_balkon_peryla_send(str_Rec:=fb_KL6301_0.str_Data_Rec, bData:=balkon_peryla,  Group_Address:=balkon_peryla_adr, bsend:=((fb_balkon_peryla_send.bData XOR fb_balkon_peryla_read.bData XOR balkon_peryla)OR fb_heartbeat2_timer.q));   (*       balkon_peryla_read.bData XOR balkon_peryla)) AND fb_heartbeat2_timer.q))      )));*)
IF NOT fb_balkon_peryla_read.bDataReceive OR  fb_heartbeat2_timer.q THEN fb_balkon_peryla_send.bSend:=FALSE; fb_balkon_peryla_send(str_Rec:=fb_KL6301_0.str_Data_Rec, bData:=balkon_peryla,  Group_Address:=balkon_peryla_adr);END_IF
fb_kino_l_send(str_Rec:=fb_KL6301_0.str_Data_Rec, bData:=kino_l,  Group_Address:=kino_l_adr, bsend:=((fb_kino_l_send.bData  <>  fb_kino_l_read.bData <> kino_l)OR fb_heartbeat2_timer.q));
IF NOT fb_kino_l_read.bDataReceive OR  fb_heartbeat2_timer.q THEN fb_kino_l_send.bSend:=FALSE; fb_kino_l_send(str_Rec:=fb_KL6301_0.str_Data_Rec,  Group_Address:=kino_l_adr);END_IF
fb_balkon_bra_send(str_Rec:=fb_KL6301_0.str_Data_Rec, bData:=balkon_bra,  Group_Address:=balkon_bra_adr, bsend:=((fb_balkon_bra_read.bData  XOR fb_balkon_bra_read.bData XOR balkon_bra)OR fb_heartbeat2_timer.q));   (*       balkon_bra_read.bData XOR balkon_bra)) AND fb_heartbeat2_timer.q))      )));*)
IF NOT fb_balkon_bra_read.bDataReceive OR  fb_heartbeat2_timer.q THEN fb_balkon_bra_send.bSend:=FALSE; fb_balkon_bra_send(str_Rec:=fb_KL6301_0.str_Data_Rec, bData:=balkon_bra,  Group_Address:=balkon_bra_adr);END_IF
fb_kabinet_balkon_l_send(str_Rec:=fb_KL6301_0.str_Data_Rec, bData:=kabinet_balkon_l,  Group_Address:=kabinet_balkon_l_adr, bsend:=(( fb_kabinet_balkon_l_send.bData XOR fb_kabinet_balkon_l_read.bData XOR kabinet_balkon_l)OR fb_heartbeat2_timer.q));   (*       kabinet_balkon_l_read.bData XOR kabinet_balkon_l)) AND fb_heartbeat2_timer.q))      )));*)
IF NOT fb_kabinet_balkon_l_read.bDataReceive OR  fb_heartbeat2_timer.q THEN fb_kabinet_balkon_l_send.bSend:=FALSE; fb_kabinet_balkon_l_send(str_Rec:=fb_KL6301_0.str_Data_Rec, bData:=kabinet_balkon_l,  Group_Address:=kabinet_balkon_l_adr);END_IF
fb_balkon_send(str_Rec:=fb_KL6301_0.str_Data_Rec, bData:=balkon,  Group_Address:=balkon_adr, bsend:=((fb_balkon_send.bData XOR fb_balkon_read.bData XOR balkon)OR fb_heartbeat2_timer.q));   (*       balkon_read.bData XOR balkon)) AND fb_heartbeat2_timer.q))      )));*)
IF NOT fb_balkon_read.bDataReceive OR  fb_heartbeat2_timer.q THEN fb_balkon_send.bSend:=FALSE; fb_balkon_send(str_Rec:=fb_KL6301_0.str_Data_Rec, bData:=balkon,  Group_Address:=balkon_adr);END_IF
fb_korydor1_send(str_Rec:=fb_KL6301_0.str_Data_Rec, bData:=korydor1,  Group_Address:=korydor1_adr, bsend:=((fb_korydor1_send.bData XOR fb_korydor1_read.bData XOR korydor1)OR fb_heartbeat2_timer.q));   (* *)
IF NOT fb_korydor1_read.bDataReceive OR  fb_heartbeat2_timer.q THEN fb_korydor1_send.bSend:=FALSE; fb_korydor1_send(str_Rec:=fb_KL6301_0.str_Data_Rec, bData:=korydor1,  Group_Address:=korydor1_adr);END_IF
fb_kino_bra_send(str_Rec:=fb_KL6301_0.str_Data_Rec, bData:=kino_bra,  Group_Address:=kino_bra_adr, bsend:=((fb_kino_bra_send.bData XOR fb_kino_bra_read.bData XOR kino_bra)OR fb_heartbeat2_timer.q));
IF NOT fb_kino_bra_read.bDataReceive OR  fb_heartbeat2_timer.q THEN fb_kino_bra_send.bSend:=FALSE; fb_kino_bra_send(str_Rec:=fb_KL6301_0.str_Data_Rec, bData:=kino_bra,  Group_Address:=kino_bra_adr);END_IF
fb_korydor2_send(str_Rec:=fb_KL6301_0.str_Data_Rec, bData:=korydor2,  Group_Address:=korydor2_adr, bsend:=((fb_korydor2_send.bData XOR fb_korydor2_read.bData XOR korydor2)OR fb_heartbeat2_timer.q));
IF NOT fb_korydor2_read.bDataReceive OR  fb_heartbeat2_timer.q THEN fb_korydor2_send.bSend:=FALSE; fb_korydor2_send(str_Rec:=fb_KL6301_0.str_Data_Rec, bData:=korydor2,  Group_Address:=korydor2_adr);END_IF
fb_studio_pidsvitka_send(str_Rec:=fb_KL6301_0.str_Data_Rec, bData:=studio_pidsvitka,  Group_Address:=studio_pidsvitka_adr, bsend:=((fb_studio_pidsvitka_send.bData XOR fb_studio_pidsvitka_read.bData XOR studio_pidsvitka)OR fb_heartbeat2_timer.q));
IF NOT fb_studio_pidsvitka_read.bDataReceive OR  fb_heartbeat2_timer.q THEN fb_studio_pidsvitka_send.bSend:=FALSE; fb_studio_pidsvitka_send(str_Rec:=fb_KL6301_0.str_Data_Rec, bData:=studio_pidsvitka,  Group_Address:=studio_pidsvitka_adr);END_IF
fb_skhody2_3_send(str_Rec:=fb_KL6301_0.str_Data_Rec, bData:=skhody2_3,  Group_Address:=skhody2_3_adr, bsend:=((fb_skhody2_3_send.bData XOR fb_skhody2_3_read.bData XOR skhody2_3)OR fb_heartbeat2_timer.q));
IF NOT fb_skhody2_3_read.bDataReceive OR  fb_heartbeat2_timer.q THEN fb_skhody2_3_send.bSend:=FALSE; fb_skhody2_3_send(str_Rec:=fb_KL6301_0.str_Data_Rec, bData:=skhody2_3,  Group_Address:=skhody2_3_adr);END_IF
fb_studio_l_send(str_Rec:=fb_KL6301_0.str_Data_Rec, bData:=studio_l,  Group_Address:=studio_l_adr, bsend:=((fb_studio_l_send.bData XOR fb_studio_l_read.bData XOR studio_l)OR fb_heartbeat2_timer.q));
IF NOT fb_studio_l_read.bDataReceive OR  fb_heartbeat2_timer.q THEN fb_studio_l_send.bSend:=FALSE; fb_studio_l_send(str_Rec:=fb_KL6301_0.str_Data_Rec, bData:=studio_l,  Group_Address:=studio_l_adr);END_IF
fb_kabinet_pidsvitka_kolo_send(str_Rec:=fb_KL6301_0.str_Data_Rec, bData:=kabinet_pidsvitka_kolo,  Group_Address:=kabinet_pidsvitka_kolo_adr, bsend:=((fb_kabinet_pidsvitka_kolo_send.bData XOR fb_kabinet_pidsvitka_kolo_read.bData XOR kabinet_pidsvitka_kolo)OR fb_heartbeat2_timer.q));
IF NOT fb_kabinet_pidsvitka_kolo_read.bDataReceive OR  fb_heartbeat2_timer.q THEN fb_kabinet_pidsvitka_kolo_send.bSend:=FALSE; fb_kabinet_pidsvitka_kolo_send(str_Rec:=fb_KL6301_0.str_Data_Rec, bData:=kabinet_pidsvitka_kolo,  Group_Address:=kabinet_pidsvitka_kolo_adr);END_IF
fb_kabinet_svitlo_send(str_Rec:=fb_KL6301_0.str_Data_Rec, bData:=kabinet_svitlo,  Group_Address:=kabinet_svitlo_adr, bsend:=((fb_kabinet_svitlo_send.bData XOR fb_kabinet_svitlo_read.bData XOR kabinet_svitlo)OR fb_heartbeat2_timer.q));
IF NOT fb_kabinet_svitlo_read.bDataReceive OR  fb_heartbeat2_timer.q THEN fb_kabinet_svitlo_send.bSend:=FALSE; fb_kabinet_svitlo_send(str_Rec:=fb_KL6301_0.str_Data_Rec, bData:=kabinet_svitlo,  Group_Address:=kabinet_svitlo_adr);END_IF
fb_stend_send(str_Rec:=fb_KL6301_0.str_Data_Rec, bData:=stend,  Group_Address:=stend_adr, bsend:=((fb_stend_send.bData XOR fb_stend_read.bData XOR stend)OR fb_heartbeat2_timer.q));
IF NOT fb_stend_read.bDataReceive OR  fb_heartbeat2_timer.q THEN fb_stend_send.bSend:=FALSE; fb_stend_send(str_Rec:=fb_KL6301_0.str_Data_Rec, bData:=stend,  Group_Address:=stend_adr);END_IF
fb_kabinet_kobra_send(str_Rec:=fb_KL6301_0.str_Data_Rec, bData:=kabinet_kobra,  Group_Address:=kabinet_kobra_adr, bsend:=((fb_kabinet_kobra_send.bData XOR fb_kabinet_kobra_read.bData XOR kabinet_kobra)OR fb_heartbeat2_timer.q));
IF NOT fb_kabinet_kobra_read.bDataReceive OR  fb_heartbeat2_timer.q THEN fb_kabinet_kobra_send.bSend:=FALSE; fb_kabinet_kobra_send(str_Rec:=fb_KL6301_0.str_Data_Rec, bData:=kabinet_kobra,  Group_Address:=kabinet_kobra_adr);END_IF
fb_skhody_peryla_send(str_Rec:=fb_KL6301_0.str_Data_Rec, bData:=skhody_peryla,  Group_Address:=skhody_peryla_adr, bsend:=((fb_skhody_peryla_send.bData XOR fb_skhody_peryla_read.bData XOR skhody_peryla)OR fb_heartbeat2_timer.q));
IF NOT fb_skhody_peryla_read.bDataReceive OR  fb_heartbeat2_timer.q THEN fb_skhody_peryla_send.bSend:=FALSE; fb_skhody_peryla_send(str_Rec:=fb_KL6301_0.str_Data_Rec, bData:=skhody_peryla,  Group_Address:=skhody_peryla_adr);END_IF
fb_tambur2_send(str_Rec:=fb_KL6301_0.str_Data_Rec, bData:=tambur2,  Group_Address:=tambur2_adr, bsend:=((fb_tambur2_send.bData XOR fb_tambur2_read.bData XOR tambur2)OR fb_heartbeat2_timer.q)) ;
IF NOT fb_tambur2_read.bDataReceive OR  fb_heartbeat2_timer.q THEN fb_tambur2_send.bSend:=FALSE; fb_tambur2_send(str_Rec:=fb_KL6301_0.str_Data_Rec, bData:=tambur2,  Group_Address:=tambur2_adr);END_IF

IF NOT  fb_balkon_peryla_read.bDataReceive THEN
	data2floor[100].0:=fb_balkon_peryla_read.bdata;
	balkon_peryla:=fb_balkon_peryla_read.bdata;
ELSE data2floor[100].0:=balkon_peryla; END_IF
IF NOT fb_kino_l_read.bDataReceive THEN
	data2floor[100].1:=fb_kino_l_read.bdata;
	kino_l:=fb_kino_l_read.bdata;
ELSE data2floor[100].1:=kino_l; END_IF
IF NOT fb_balkon_bra_read.bDataReceive THEN
	data2floor[100].2:= fb_balkon_bra_read.bdata;
	balkon_bra:= fb_balkon_bra_read.bdata;
ELSE data2floor[100].2:= balkon_bra;END_IF
IF NOT fb_kabinet_balkon_l_read.bDataReceive  THEN
	 data2floor[100].3:=fb_kabinet_balkon_l_read.bdata;
	kabinet_balkon_l:=fb_kabinet_balkon_l_read.bdata;
ELSE 	data2floor[100].3:=kabinet_balkon_l; END_IF
IF NOT fb_balkon_read.bDataReceive THEN
	data2floor[100].4:=fb_balkon_read.bdata;
	balkon:=fb_balkon_read.bdata;
ELSE 	data2floor[100].4:=balkon; END_IF
IF NOT fb_korydor1_read.bDataReceive THEN
	data2floor[100].5:=fb_korydor1_read.bdata;
	korydor1:=fb_korydor1_read.bdata;
ELSE 	data2floor[100].5:=korydor1;END_IF;
IF NOT fb_kino_bra_read.bDataReceive  THEN
	data2floor[100].6:=fb_kino_bra_read.bdata;
	kino_bra:=fb_kino_bra_read.bdata;
 ELSE 	data2floor[100].6:=kino_bra; END_IF;
IF NOT fb_korydor2_read.bDataReceive  THEN
	data2floor[100].7:=fb_korydor2_read.bdata;
	korydor2:=fb_korydor2_read.bdata;
ELSE 	data2floor[100].7:=korydor2; END_IF;
IF NOT fb_studio_pidsvitka_read.bDataReceive  THEN
	data2floor[101].0:=fb_studio_pidsvitka_read.bdata;
	studio_pidsvitka:=fb_studio_pidsvitka_read.bdata;
ELSE data2floor[101].0:=studio_pidsvitka; END_IF;
IF NOT fb_skhody2_3_read.bDataReceive  THEN
	data2floor[101].1:=fb_skhody2_3_read.bdata;
	skhody2_3:=fb_skhody2_3_read.bdata;
ELSE data2floor[101].1:=skhody2_3; END_IF;
IF NOT fb_studio_l_read.bDataReceive THEN
	data2floor[101].2:=fb_studio_l_read.bdata;
	studio_l:=fb_studio_l_read.bdata;
ELSE data2floor[101].2:=studio_l; END_IF;
IF NOT fb_kabinet_pidsvitka_kolo_read.bDataReceive THEN
	data2floor[101].3:=fb_kabinet_pidsvitka_kolo_read.bdata;
	kabinet_pidsvitka_kolo:=fb_kabinet_pidsvitka_kolo_read.bdata;
ELSE data2floor[101].3:=kabinet_pidsvitka_kolo; END_IF;
IF NOT fb_kabinet_svitlo_read.bDataReceive THEN
	data2floor[101].4:=fb_kabinet_svitlo_read.bdata;
	kabinet_svitlo:=fb_kabinet_svitlo_read.bdata;
ELSE data2floor[101].4:=kabinet_svitlo; END_IF;
IF NOT fb_kabinet_kobra_read.bDataReceive THEN
	data2floor[101].5:=fb_kabinet_kobra_read.bdata;
	kabinet_kobra:=fb_kabinet_kobra_read.bdata;
ELSE data2floor[101].5:=kabinet_kobra; END_IF;
IF NOT fb_tambur2_read.bDataReceive  THEN
	data2floor[101].6:=fb_tambur2_read.bdata;
	tambur2:=fb_tambur2_read.bdata;
ELSE data2floor[101].6:=tambur2; END_IF;
IF NOT fb_stend_read.bDataReceive  THEN
	data2floor[101].7:=fb_stend_read.bdata;
	stend:=fb_stend_read.bdata;
ELSE  data2floor[101].7:=stend; END_IF;
IF NOT fb_skhody_peryla_read.bDataReceive  THEN
	data2floor[102].0:=fb_skhody_peryla_read.bdata;
	skhody_peryla:=fb_skhody_peryla_read.bdata;
ELSE data2floor[102].0:=skhody_peryla; END_IF;
END_ACTION

(* POU ADS_write, ST *)
PROGRAM ADS_write
VAR
	write_timeout: TIME;
	b_write1, b_write2: BOOL;
	write_ads1, write_ads2, write_ads4: ADSWRITE;

	timer1, timer2:TP;
	errorcounter1, errorcounter2, pack_c:CTU ;
	test_word: WORD;
	i,j,i1,j1, i4,j4: INT;
	data_changed: BOOL;
	try_again2, try_again1, try_again4: BOOL;
	timer4: TP;
	b_write4: BOOL;
	errorcounter4: CTU;
END_VAR
write_timeout:=t#3s;

FOR i:=0 TO (SIZEOF(data2floor))-1 DO
	IF data2floor[i]<>data2floor_prev[i]  OR try_again2 THEN
		b_write2:=TRUE;
		EXIT;
	ELSE
		b_write2:=FALSE;
	END_IF
END_FOR

IF write_ads2.BUSY THEN b_write2:=FALSE; END_IF

	write_ads2(
		NETID:=ads_adr2,
		PORT:=800,
		IDXGRP:=16#4020,
		IDXOFFS:=300,
		WRITE:=b_write2,
		TMOUT:=write_timeout,
		LEN:=SIZEOF(data2floor),
		SRCADDR:=ADR(data2floor));
write_ads2.WRITE:=FALSE;

IF write_ads2.ERR AND NOT timer2.Q THEN
	timer2.IN:=TRUE;
	try_again2:=TRUE;
ELSE try_again2:=FALSE;
END_IF
timer2(PT:=write_timeout*2);
timer2.IN:=FALSE;


FOR j:=0 TO (SIZEOF(data2floor))-1 DO
	data2floor_prev[j]:=data2floor[j];
END_FOR

(*1floor*)
FOR i1:=0 TO (SIZEOF(data1floor))-1 DO
	IF data1floor[i1]<>data1floor_prev[i1] AND NOT timer1.Q THEN
		b_write1:=TRUE;
		EXIT;
	ELSE
		b_write1:=FALSE;
	END_IF
END_FOR

IF try_again1 AND NOT timer1.Q THEN
	b_write1:=TRUE;
	try_again1:=FALSE;
END_IF

errorcounter1(cu:=write_ads1.ERR);


IF write_ads1.BUSY THEN b_write1:=FALSE; END_IF

	write_ads1(
		NETID:=ads_adr1,
		PORT:=800,
		IDXGRP:=16#4020,
		IDXOFFS:=300,
		WRITE:=b_write1,
		TMOUT:=write_timeout,
		LEN:=SIZEOF(data1floor),
		SRCADDR:=ADR(data1floor));

IF write_ads1.ERR AND NOT timer1.Q THEN
	timer1.IN:=TRUE;
	try_again1:=TRUE;
END_IF
timer1(PT:=write_timeout);
timer1.IN:=FALSE;


FOR j1:=0 TO (SIZEOF(data1floor))-1 DO
	data1floor_prev[j1]:=data1floor[j1];
END_FOR

(*derevo*)
FOR i4:=0 TO (SIZEOF(data_derevo))-1 DO
	IF data_derevo[i4]<>data_derevo_prev[i4] AND NOT timer4.Q THEN
		b_write4:=TRUE;
		EXIT;
	ELSE
		b_write4:=FALSE;
	END_IF
END_FOR

IF try_again4 AND NOT timer4.Q THEN
	b_write4:=TRUE;
	try_again4:=FALSE;
END_IF

errorcounter4(cu:=write_ads4.ERR);


IF write_ads4.BUSY THEN b_write4:=FALSE; END_IF

	write_ads4(
		NETID:=ads_adr4,
		PORT:=800,
		IDXGRP:=16#4020,
		IDXOFFS:=400,
		WRITE:=b_write4,
		TMOUT:=write_timeout,
		LEN:=SIZEOF(data_derevo),
		SRCADDR:=ADR(data_derevo));

IF write_ads4.ERR AND NOT timer4.Q THEN
	timer4.IN:=TRUE;
	try_again4:=TRUE;
END_IF
timer4(PT:=write_timeout);
timer4.IN:=FALSE;


FOR j4:=0 TO (SIZEOF(data_derevo))-1 DO
	data_derevo_prev[j4]:=data_derevo[j4];
END_FOR
END_PROGRAM

(* POU HVAC/winter, ST *)
PROGRAM winter
VAR

END_VAR
(*1-COOL mode 2-HEAT mode, 3-FAN mode*)

(*--------------------------VITALNYA---------------------------------------------------------------*)

	IF VITALNYA_HVAC.heat_mode=2 THEN
				VITALNYA_HVAC.zaslinka:=TRUE;(*closed*)
				VITALNYA_HVAC.tepla_pidloga:=TRUE; (*all opened*)
		CASE VITALNYA_HVAC.heat_speed OF

			1:	VITALNYA_HVAC.fancoil_speed:=1;
				VITALNYA_HVAC.klapan:=16#3FFF;
			2:	VITALNYA_HVAC.fancoil_speed:=2;
				VITALNYA_HVAC.klapan:=16#5FFF;
			3:	VITALNYA_HVAC.fancoil_speed:=3;
				VITALNYA_HVAC.klapan:=16#7FFF;
		END_CASE
	END_IF

	IF VITALNYA_HVAC.heat_mode=1 THEN
				VITALNYA_HVAC.klapan:=16#0;(*full closed*)
				VITALNYA_HVAC.zaslinka:=FALSE;
				VITALNYA_HVAC.tepla_pidloga:=FALSE; (*all closed*)

			CASE VITALNYA_HVAC.heat_speed OF
			1:	VITALNYA_HVAC.fancoil_speed:=1;
			2:	VITALNYA_HVAC.fancoil_speed:=2;
			3:	VITALNYA_HVAC.fancoil_speed:=3;
		END_CASE
	END_IF

	IF VITALNYA_HVAC.heat_mode=3 THEN
		VITALNYA_HVAC.tepla_pidloga:=FALSE;
		IF heat.t_out<0 THEN VITALNYA_HVAC.klapan:=16#3FFF;(*30%*) ELSE VITALNYA_HVAC.klapan:=16#0;END_IF
		CASE VITALNYA_HVAC.heat_speed OF
			1:	VITALNYA_HVAC.fancoil_speed:=0;
				VITALNYA_HVAC.zaslinka:=TRUE;(*closed*)
				VITALNYA_HVAC.klapan:=16#0;(*full closed*)
			2:	VITALNYA_HVAC.fancoil_speed:=2;
				VITALNYA_HVAC.zaslinka:=FALSE;(*opened*)
			3:	VITALNYA_HVAC.fancoil_speed:=3;
				VITALNYA_HVAC.zaslinka:=FALSE;(*opened*)
		END_CASE
	END_IF



(*--------------------------KABINET---------------------------------------------------------------*)
(*реверс двигуна клапана*)

	IF KABINET_HVAC.heat_mode=2 THEN
				KABINET_HVAC.zaslinka:=TRUE;(*closed*)
				KABINET_HVAC.tepla_pidloga:=TRUE; (*all opened*)
		CASE KABINET_HVAC.heat_speed OF

			1:	KABINET_HVAC.fancoil_speed:=1;
				KABINET_HVAC.klapan:=16#5FFF;
			2:	KABINET_HVAC.fancoil_speed:=2;
				KABINET_HVAC.klapan:=16#3FFF;
			3:	KABINET_HVAC.fancoil_speed:=3;
				KABINET_HVAC.klapan:=16#1FFF;
		END_CASE
	END_IF

	IF KABINET_HVAC.heat_mode=1 THEN
				KABINET_HVAC.klapan:=16#7FFF;(*full closed*)
				KABINET_HVAC.zaslinka:=FALSE;
				KABINET_HVAC.tepla_pidloga:=FALSE; (*all closed*)

			CASE KABINET_HVAC.heat_speed OF
			1:	KABINET_HVAC.fancoil_speed:=1;
			2:	KABINET_HVAC.fancoil_speed:=2;
			3:	KABINET_HVAC.fancoil_speed:=3;
		END_CASE
	END_IF

	IF KABINET_HVAC.heat_mode=3 THEN
		KABINET_HVAC.tepla_pidloga:=FALSE;
		IF heat.t_out<0 THEN KABINET_HVAC.klapan:=16#5FFF;(*30%*) ELSE KABINET_HVAC.klapan:=16#7FFF;END_IF
		CASE KABINET_HVAC.heat_speed OF
			1:	KABINET_HVAC.fancoil_speed:=0;
				KABINET_HVAC.zaslinka:=TRUE;(*closed*)
				KABINET_HVAC.klapan:=16#7FFF;(*full closed*)
			2:	KABINET_HVAC.fancoil_speed:=2;
				KABINET_HVAC.zaslinka:=FALSE;(*opened*)
			3:	KABINET_HVAC.fancoil_speed:=3;
				KABINET_HVAC.zaslinka:=FALSE;(*opened*)
		END_CASE
	END_IF



(*--------------------------KINO---------------------------------------------------------------*)
(*реверс двигуна клапана*)
	IF KINO_HVAC.heat_mode=2 THEN
				KINO_HVAC.zaslinka:=TRUE;(*closed*)
				KINO_HVAC.tepla_pidloga:=TRUE; (*all opened*)
		CASE KINO_HVAC.heat_speed OF

			1:	KINO_HVAC.fancoil_speed:=1;
				KINO_HVAC.klapan:=16#5FFF;
			2:	KINO_HVAC.fancoil_speed:=2;
				KINO_HVAC.klapan:=16#3FFF;
			3:	KINO_HVAC.fancoil_speed:=3;
				KINO_HVAC.klapan:=16#1FFF;
		END_CASE
	END_IF

	IF KINO_HVAC.heat_mode=1 THEN
				KINO_HVAC.klapan:=16#0;(*full closed*)
				KINO_HVAC.zaslinka:=FALSE;
				KINO_HVAC.tepla_pidloga:=FALSE; (*all closed*)

			CASE KINO_HVAC.heat_speed OF
			1:	KINO_HVAC.fancoil_speed:=1;
			2:	KINO_HVAC.fancoil_speed:=2;
			3:	KINO_HVAC.fancoil_speed:=3;
		END_CASE
	END_IF

	IF KINO_HVAC.heat_mode=3 THEN
		KINO_HVAC.tepla_pidloga:=FALSE;
		IF heat.t_out<0 THEN KINO_HVAC.klapan:=16#5FFF;(*30%*) ELSE KINO_HVAC.klapan:=16#7FFF;END_IF
		CASE KINO_HVAC.heat_speed OF
			1:	KINO_HVAC.fancoil_speed:=0;
				KINO_HVAC.zaslinka:=TRUE;(*closed*)
				KINO_HVAC.klapan:=16#7FFF;(*full closed*)
			2:	KINO_HVAC.fancoil_speed:=2;
				KINO_HVAC.zaslinka:=FALSE;(*opened*)
			3:	KINO_HVAC.fancoil_speed:=3;
				KINO_HVAC.zaslinka:=FALSE;(*opened*)
		END_CASE
	END_IF



(*--------------------------DYTJACHA---------------------------------------------------------------*)
(*реверс двигуна клапана*)
	IF DYTJACHA_HVAC.heat_mode=2 THEN
				DYTJACHA_HVAC.zaslinka:=TRUE;(*closed*)
				DYTJACHA_HVAC.tepla_pidloga:=TRUE; (*all opened*)
		CASE DYTJACHA_HVAC.heat_speed OF

			1:	DYTJACHA_HVAC.fancoil_speed:=1;
				DYTJACHA_HVAC.klapan:=16#5FFF;
			2:	DYTJACHA_HVAC.fancoil_speed:=2;
				DYTJACHA_HVAC.klapan:=16#3FFF;
			3:	DYTJACHA_HVAC.fancoil_speed:=3;
				DYTJACHA_HVAC.klapan:=16#1FFF;
		END_CASE
	END_IF

	IF DYTJACHA_HVAC.heat_mode=1 THEN
				DYTJACHA_HVAC.klapan:=16#7FFF;(*full closed*)
				DYTJACHA_HVAC.zaslinka:=FALSE;
				DYTJACHA_HVAC.tepla_pidloga:=FALSE; (*all closed*)

			CASE DYTJACHA_HVAC.heat_speed OF
			1:	DYTJACHA_HVAC.fancoil_speed:=1;
			2:	DYTJACHA_HVAC.fancoil_speed:=2;
			3:	DYTJACHA_HVAC.fancoil_speed:=3;
		END_CASE
	END_IF

	IF DYTJACHA_HVAC.heat_mode=3 THEN
		DYTJACHA_HVAC.tepla_pidloga:=FALSE;
		IF heat.t_out<0 THEN DYTJACHA_HVAC.klapan:=16#5FFF;(*30%*) ELSE DYTJACHA_HVAC.klapan:=16#7FFF;END_IF
		CASE DYTJACHA_HVAC.heat_speed OF
			1:	DYTJACHA_HVAC.fancoil_speed:=0;
				DYTJACHA_HVAC.zaslinka:=TRUE;(*closed*)
				DYTJACHA_HVAC.klapan:=16#7FFF;(*full closed*)
			2:	DYTJACHA_HVAC.fancoil_speed:=2;
				DYTJACHA_HVAC.zaslinka:=FALSE;(*opened*)
			3:	DYTJACHA_HVAC.fancoil_speed:=3;
				DYTJACHA_HVAC.zaslinka:=FALSE;(*opened*)
		END_CASE
	END_IF



(*--------------------------SPALNYA---------------------------------------------------------------*)

	IF SPALNYA_HVAC.heat_mode=2 THEN
				SPALNYA_HVAC.zaslinka:=TRUE;(*closed*)
				SPALNYA_HVAC.tepla_pidloga:=TRUE; (*all opened*)
		CASE SPALNYA_HVAC.heat_speed OF

			1:	SPALNYA_HVAC.fancoil_speed:=1;
				SPALNYA_HVAC.klapan:=16#3FFF;
			2:	SPALNYA_HVAC.fancoil_speed:=2;
				SPALNYA_HVAC.klapan:=16#5FFF;
			3:	SPALNYA_HVAC.fancoil_speed:=3;
				SPALNYA_HVAC.klapan:=16#7FFF;
		END_CASE
	END_IF

	IF SPALNYA_HVAC.heat_mode=1 THEN
				SPALNYA_HVAC.klapan:=16#0;(*full closed*)
				SPALNYA_HVAC.zaslinka:=FALSE;
				SPALNYA_HVAC.tepla_pidloga:=FALSE; (*all closed*)

			CASE SPALNYA_HVAC.heat_speed OF
			1:	SPALNYA_HVAC.fancoil_speed:=1;
			2:	SPALNYA_HVAC.fancoil_speed:=2;
			3:	SPALNYA_HVAC.fancoil_speed:=3;
		END_CASE
	END_IF

	IF SPALNYA_HVAC.heat_mode=3 THEN
		SPALNYA_HVAC.tepla_pidloga:=FALSE;
		IF heat.t_out<0 THEN SPALNYA_HVAC.klapan:=16#3FFF;(*30%*) ELSE SPALNYA_HVAC.klapan:=16#0;END_IF
		CASE SPALNYA_HVAC.heat_speed OF
			1:	SPALNYA_HVAC.fancoil_speed:=0;
				SPALNYA_HVAC.zaslinka:=TRUE;(*closed*)
				SPALNYA_HVAC.klapan:=16#0;(*full closed*)
			2:	SPALNYA_HVAC.fancoil_speed:=2;
				SPALNYA_HVAC.zaslinka:=FALSE;(*opened*)
			3:	SPALNYA_HVAC.fancoil_speed:=3;
				SPALNYA_HVAC.zaslinka:=FALSE;(*opened*)
		END_CASE
	END_IF
END_PROGRAM
